(* IEC 61131-3 sources: HappyLearnCodesys/content/softmotion/BasicMotion_GearInPos, 4 files *)

(* ---- GVL_Const.st ---- *)
/// 本全域常數表定義輸送帶、工件與鋸片工具的幾何尺寸與同步位置，供 BasicMotion_GearInPos 範例的所有程式共用。
{attribute 'qualified_only'}
VAR_GLOBAL CONSTANT
    /// 鋸片與工件同步時的 X 座標位置。
    SYNCPOS : LREAL := 0;

    /// 光遮斷器在輸送帶座標系下的 X 座標位置。
    LIGHTBARRIERPOS : LREAL := -300;

    /// 工件的幾何尺寸（長、寬、高，單位 mm）。
    WORKPIECELENGTH : LREAL := 200;
    WORKPIECEWIDTH : LREAL := 120;
    WORKPIECEHEIGHT : LREAL := 10;

    /// 輸送帶的外觀尺寸（長、寬、高，單位 mm）。
    BELTLENGTH : LREAL:= 1000;
    BELTWIDTH : LREAL:= 150;
    BELTHEIGHT : LREAL:= 50;

    /// 鋸片切削端相對於連桿末端的偏移距離（單位 mm）。
    TIPOFFSET : LREAL := 8 ;
END_VAR

(* ---- DepictorCalculation.st ---- *)
/// 此程式負責將輸送帶的幾何形狀與當前位置轉換成可視化元件，供 3D/2D 視覺化畫面使用。
/// 透過 BeltDepictor 功能塊與 Master 軸的位置，讓使用者在視覺化畫面上看到輸送帶隨 Master 軸移動。
PROGRAM DepictorCalculation
VAR
    /// 表示輸送帶外觀與位置的描繪功能塊。
    beltFB : BeltDepictor :=
        (posOrigin:= (dX:= 0, dY:= 0, dZ:= 0),
         length:= Const.BELTLENGTH,
         width:= Const.BELTWIDTH,
         height:= Const.BELTHEIGHT);
END_VAR

/// 以 Master 軸的實際位置驅動描繪功能塊，更新輸送帶在畫面上的位置。
beltFB(beltPos:= Master.fSetPosition);

(* ---- PLC_PRG.st ---- *)
/// 這是 GearInPos 範例的主控程式，負責：
/// 1. 啟動三個軸（Master 輸送帶軸、Slave 鋸片滑台軸、Tool 刀具上下軸）的伺服驅動。
/// 2. 以固定速度驅動輸送帶（Master 軸）前進。
/// 3. 在光遮斷器偵測到工件後，利用 MC_GearInPos 讓鋸片滑台（Slave 軸）在指定位置與輸送帶同步。
/// 4. 控制刀具（Tool 軸）完成一次切割動作，並將鋸片滑台與刀具移回安全待命位置。
PROGRAM PLC_PRG
VAR
    /// 控制 Tool 軸（刀具上下移動）的電源功能塊。
    pwTool   : MC_Power := (bRegulatorOn:= TRUE, bDriveStart:= TRUE);
    /// 控制 Master 軸（輸送帶）的電源功能塊。
    pwMaster : MC_Power := (bRegulatorOn:= TRUE, bDriveStart:= TRUE);
    /// 控制 Slave 軸（鋸片滑台）的電源功能塊。
    pwSlave  : MC_Power := (bRegulatorOn:= TRUE, bDriveStart:= TRUE);

    /// 用於在指定位置讓 Slave 軸與 Master 軸進行齒輪同步的功能塊。
    gearInPos: MC_GearInPos := (
         RatioNumerator:= 1,
         RatioDenominator:= 1);

    /// 控制輸送帶（Master 軸）以固定速度運轉的速度模式運動命令。
	moveBelt : MC_MoveVelocity := (
        Velocity:= 250,
        Acceleration:= 500,
        Deceleration:= 500,
        Jerk:= 5000);

    /// 控制刀具（Tool 軸）上下移動的絕對位置運動命令。
    moveTool : MC_MoveAbsolute := (
        Velocity:= 500,
        Acceleration:= 10000,
        Deceleration:= 10000,
        Jerk:= 200000) ;

    /// 控制鋸片滑台（Slave 軸）回到待命位置的絕對位置運動命令。
    moveSlave : MC_MoveAbsolute := (
        Velocity:= 400,
        Acceleration:= 5000,
        Deceleration:= 5000,
        Jerk:= 100000) ;

    /// 主狀態機，決定目前處於哪一個控制階段。
	state : UDINT;
END_VAR
VAR CONSTANT
	/// 軸上電與伺服準備階段。
	STATE_POWER : UDINT := 0;
	/// 等待工件被光遮斷器偵測到。
	STATE_WAIT_FOR_WORKPIECE : UDINT := 10;
    /// 已下達 GearInPos 命令，等待 Master 與 Slave 軸真正進入同步。
    STATE_WAIT_FOR_SYNC : UDINT := 20;
    /// 刀具由原點移動到切削位置。
    STATE_MOVE_TOOL_0 : UDINT := 30;
    /// 刀具由切削位置返回原點。
    STATE_MOVE_TOOL_1 : UDINT := 40;
    /// 鋸片滑台回到待命位置。
    STATE_MOVE_TO_REST : UDINT := 50;
END_VAR

/// 依照不同狀態執行對應的軸控制與命令切換。
CASE state OF
STATE_POWER:
    /// 依序啟動三個軸的電源與驅動，等待皆準備就緒。
    pwTool.Enable := TRUE;
    pwMaster.Enable := TRUE;
    pwSlave.Enable := TRUE;

    IF pwTool.Status AND pwMaster.Status AND pwSlave.Status
    THEN
        /// 當三個軸皆就緒後，啟動輸送帶以固定速度前進，並進入等待工件的狀態。
        moveBelt.Execute := TRUE;
        state := STATE_WAIT_FOR_WORKPIECE;
    END_IF

STATE_WAIT_FOR_WORKPIECE:
    /// 一旦模擬程式回報偵測到工件，即準備計算齒輪同步的關鍵位置。
    IF SimulateWorkpiece.WorkpieceDetected THEN
        /// MasterSyncPosition：以目前 Master 位置為基準，再加上工件從光遮斷器到同步點的距離，
        ///                     並略為提前 10% 工件長度，讓切割動作在工件進入同步位置前啟動。
        gearInPos.MasterSyncPosition := Master.fSetPosition + (Const.SYNCPOS - Const.LIGHTBARRIERPOS) + Const.WORKPIECELENGTH*0.1;
        /// SlaveSyncPosition：Slave 軸達到此位置時，即與 Master 軸進入同步狀態。
        gearInPos.SlaveSyncPosition:= Const.SYNCPOS;
        /// MasterStartDistance：當 Master 再前進一定距離後才真正執行齒輪同步，避免命令一下達就立即啟動。
        gearInPos.MasterStartDistance := 0.75*(Const.SYNCPOS - Const.LIGHTBARRIERPOS);
        /// 下達齒輪同步命令，進入等待同步完成的狀態。
        gearInPos.Execute := TRUE;
        state := STATE_WAIT_FOR_SYNC;
    END_IF

STATE_WAIT_FOR_SYNC:
    /// 當 GearInPos 回報已進入同步狀態，代表鋸片滑台與輸送帶已對齊。
    IF gearInPos.InSync THEN
        /// 將刀具移至帶寬加上刀尖偏移的位置，模擬切入工件。
        moveTool.Position := Const.BELTWIDTH + Const.TIPOFFSET;
        moveTool.Execute := TRUE;
        state := STATE_MOVE_TOOL_0;
    END_IF

STATE_MOVE_TOOL_0:
    /// 刀具到達切削位置後，關閉 Execute，準備指令返回原點。
    IF moveTool.Done THEN
        moveTool.Execute := FALSE;
        state := STATE_MOVE_TOOL_1;
    END_IF

STATE_MOVE_TOOL_1:
    /// 將刀具目標位置設回 0（原點），啟動回程。
    moveTool.Position := 0;
    moveTool.Execute := TRUE;

    IF moveTool.Done THEN
        /// 切割動作完成後，關閉齒輪同步與刀具運動命令，
        /// 再讓鋸片滑台移往較安全的待命位置。
        gearInPos.Execute := FALSE;
        moveTool.Execute := FALSE;
        moveSlave.Execute := TRUE;
        moveSlave.Position := 0.5*(Const.SYNCPOS + Const.LIGHTBARRIERPOS);
        state := STATE_MOVE_TO_REST;
    END_IF

STATE_MOVE_TO_REST:
    /// 鋸片滑台回到待命位置後，關閉命令並回到等待下一塊工件的狀態。
    IF moveSlave.Done THEN
        moveSlave.Execute := FALSE;
        state := STATE_WAIT_FOR_WORKPIECE ;
    END_IF
END_CASE

/// 將電源功能塊實際連接到三個軸上。
pwTool(Axis:= Tool);
pwMaster(Axis:= Master);
pwSlave(Axis:= Slave);

/// 持續以速度模式驅動輸送帶（Master 軸）。
moveBelt(Axis:= Master);

/// 在 Master 與 Slave 之間建立齒輪同步關係。
gearInPos(Master:= Master, Slave:= Slave);

/// 控制刀具與鋸片滑台的點到點移動。
moveTool(Axis:= Tool);
moveSlave(Axis:= Slave);

(* ---- SimulateWorkpiece.st ---- *)
/// 此程式負責在沒有實體感測器與工件的情況下，模擬一塊工件在輸送帶上移動，
/// 並依據工件與光遮斷器的相對位置，輸出「是否偵測到工件」的訊號與工件中心位置。
PROGRAM SimulateWorkpiece
VAR_INPUT
    /// 光遮斷器在輸送帶座標系下的 X 位置（單位 mm）。
    LightBarrierPos : LREAL := Const.LIGHTBARRIERPOS ;
    /// 工件的長度（單位 mm）。
    WorkpieceLength : LREAL := CONST.WORKPIECELENGTH ;
END_VAR
VAR_OUTPUT
    /// 當工件經過光遮斷器時，此輸出為 TRUE。
    WorkpieceDetected : BOOL ;
    /// 工件中心在輸送帶座標系下的 X 位置。
    WorkPiecePos : LREAL ;
END_VAR
VAR
    /// 工件模擬的狀態機，目前是「初始化」或「工件運行中」。
    state : UDINT;
    /// 用來記錄 Master 軸在工件產生當下的位置，用於處理位置換算與週期性回捲。
    masterOffset : LREAL;
END_VAR
VAR CONSTANT
    /// 初始化狀態：產生一塊新的工件並重設位置。
    STATE_INIT : UDINT := 0;
    /// 工件正在輸送帶上移動的狀態。
    STATE_WORKPIECE_ACTIVE : UDINT := 10;
END_VAR

/// 依狀態機決定工件當前位置與是否需要重新產生工件。
CASE state OF
STATE_INIT:
    /// 將工件中心放在輸送帶左端外側，準備讓輸送帶帶動工件往右移動。
    WorkPiecePos := -Const.BELTLENGTH/2;
    /// 記錄此時 Master 軸的位置，作為後續換算的基準點。
    masterOffset := Master.fSetPosition;
    /// 進入工件運行狀態。
    state := STATE_WORKPIECE_ACTIVE;

STATE_WORKPIECE_ACTIVE:
    /// 若 Master 軸位置因為週期性回捲而小於基準值，將基準值往回平移一個週期，維持連續位移。
    IF Master.fSetPosition < masterOffset THEN
        masterOffset := masterOffset - Master.fPositionPeriod ;
    END_IF

    /// 依 Master 軸位移量計算工件中心在輸送帶上的實際位置。
    WorkPiecePos := -Const.BELTLENGTH/2 + (Master.fSetPosition - masterOffset);

    /// 當工件通過輸送帶右端（加上一半工件長度）時，重新回到初始化狀態，準備下一塊工件。
    IF WorkPiecePos >= Const.BELTLENGTH/2 - WorkpieceLength/2 THEN
        state := STATE_INIT;
    END_IF
END_CASE

/// 當工件區間覆蓋到光遮斷器位置時，即視為「感測到工件」。
WorkpieceDetected :=
    WorkPiecePos - WorkpieceLength/2 <= LightBarrierPos AND
    WorkPiecePos + WorkpieceLength/2 >= LightBarrierPos;
